(* CODESYS project HowToUse_MIC7001_baselib.2020.0527.1.project

Project tree, tasks and I/O mapping:
  Device : Changsha-Cyber-MI-linux, Changsha Cyber-MI Co., Ltd., version 3.5.10.40
    application Application
      libraries: Standard, * (System); SysFile, 3.5.15.0 (System); SysTypes2 Interfaces, * (System); SysShm, * (System); CAA Mathematics, * (CAA Technical Workgroup); SysTime, 3.5.9.0 (System); CAA Types Extern, 3.5.13.0 (CAA Technical Workgroup); CAA DTUtil Extern, 3.5.12.0 (CAA Technical Workgroup); Util, * (System); TCP, 3.5.15.0 (3S - Smart Software Solutions GmbH); CAA Net Base Services, 3.5.15.0 (CAA Technical Workgroup); MIC7001 base library, 0.93 (Cyber-MI.com); CAA SerialCom, 3.5.15.0 (CAA Technical Workgroup)
      task task_fast (cyclic, interval 20 ms, priority 10, watchdog 300 ms x 10) calls prg_data2file, prg_others
      task task_middle (cyclic, interval 100 ms, priority 20, watchdog 500 ms x 5) calls prg_mqtt
      task task_slow (cyclic, interval 500 ms, priority 30, watchdog 900 ms x 10) calls prg_retain, prg_set_inmode
      Enums/
        data type ERROR
        data type MQTT_STATE
        data type UDP_STATE_1
      data type UDP_STATE
      programs/
        program prg_set_inmode [CFC]
        program prg_data2file [ST]
        program prg_retain [ST]
        program prg_mqtt [CFC]: ACT_boot, ACT_publish, ACT_recv_proc, ACT_first_buffer, ACT_normal_buffer, ACT_running_light, proc_get_command, proc_set_command, find_key
        program prg_others [ST]
    SoftMotion General Axis Pool
    IoDrvMIC7001 : IoDrvMIC7001, Cyber-MI, version 19.1.1
        output Application.prg_others.ao_00 : DWORD  // Ao00-Ai46@C22
        output Application.prg_others.ao_01 : DWORD  // Ao01-Ai47@D14
        output Application.prg_others.led_run : BOOL  // LED_run
        output Application.prg_others.led_run : BOOL  // LED_usr
        unmapped channels: Ai00@C16, Ai01@C28, Ai02@C17, Ai03@C29, Ai04@C30, Ai05@C19, Ai06@C31, Ai07@C20, Ai08@C18, Ai09@D18, Ai10@D20, Ai11@D31, Ai12@D19, Ai13@D30, Ai14@D29, Ai15@D17, Ai16@D28, Ai17@D16, Ai18-Do00@C25, Ai19-Do01@C24, Ai20-Do02@C13, Ai21-Do03@C01, Ai22-Do04@C03, Ai23-Do05@C04, Ai24-Do06@C05, Ai25-Do07@C06, Ai26-Do08@C08, Ai27-Do09@C09, Ai28-Do10@C10, Ai29-Do11@C11, Ai30-Do12@D34, Ai31-Do13@D35, Ai32-Do14@D23, Ai33-Do15@D12, Ai34-Do16@D10, Ai35-Do17@D09, Ai36-Do18@D08, Ai37-Do19@D07, Ai38-Do20@D05, Ai39-Do21@D04,
          Ai40-Do22@D03, Ai41-Do23@D02, Ai42-Do24@C23, Ai43-Do25@C35, Ai44-Do26@D24, Ai45-Do27@D13, Ai46-Ao00@C22, Ai47-Ao01@D14, Ai48_Pi02, Ai49_Out5V, Ai50_VCC, Ai51_VCC_L, Ai52_VCC_R, Ai53_Pwm-i0, Ai54_Pwm-i1, Ai55_Pwm-i2, Ai56_Pwm-i3, Ai57_CPU-T, Ai58_G-x, Ai59_G-y, Ai60_G-z, Ai61-reserved, Ai62-IO-cntr, Ai63-CDS-cntr, Di00-Ai00@C16, Di01-Ai01@C28, Di02-Ai02@C17, Di03-Ai03@C29, Di04-Ai04@C30, Di05-Ai05@C19, Di06-Ai06@C31, Di07-Ai07@C20, Di08-Ai08@C18, Di09-Ai09@D18, Di10-Ai10@D20, Di11-Ai11@D31, Di12-Ai12@D19, Di13-Ai13@D30, Di14-Ai14@D29, Di15-Ai15@D17,
          Di16-Ai16@D28, Di17-Ai17@D16, Di18-Ai18@C25, Di19-Ai19@C24, Di20-Ai20@C13, Di21-Ai21@C01, Di22-Ai22@C03, Di23-Ai23@C04, Di24-Ai24@C05, Di25-Ai25@C06, Di26-Ai26@C08, Di27-Ai27@C09, Di28-Ai28@C10, Di29-Ai29@C11, Di30-Ai30@D34, Di31-Ai31@D35, Di32-Ai32@D23, Di33-Ai33@D12, Di34-Ai34@D10, Di35-Ai35@D09, Di36-Ai36@D08, Di37-Ai37@D07, Di38-Ai38@D05, Di39-Ai39@D04, Di40-Ai40@D03, Di41-Ai41@D02, Di42-Ai42@C23, Di43-Ai43@C35, Di44-Ai44@D24, Di45-Ai45@D13, Di46-Ai46@C22, Di47-Ai47@D14, Di48-Pi00@C15, Di49-Pi01@C14, Di50-Pi02@D22, Di51-Pi03@D21, Di52-reserved, Di53-reserved, Di54-reserved, Di55-reserved,
          Di56-reserved, Di57-reserved, Di58-reserved, Di59-reserved, Di60-reserved, Di61-reserved, Di62-reserved, Di63-reserved, Pi00-Di48@C15, Pi01-Di49@C14, Pi02-Di50@D22, Pi03-Di51@D21, Do00-Ai18@C25, Do01-Ai19@C24, Do02-Ai20@C13, Do03-Ai21@C01, Do04-Ai22@C03, Do05-Ai23@C04, Do06-Ai24@C05, Do07-Ai25@C06, Do08-Ai26@C08, Do09-Ai27@C09, Do10-Ai28@C10, Do11-Ai29@C11, Do12-Ai30@D34, Do13-Ai31@D35, Do14-Ai32@D23, Do15-Ai33@D12, Do16-Ai34@D10, Do17-Ai35@D09, Do18-Ai36@D08, Do19-Ai37@D07, Do20-Ai38@D05, Do21-Ai39@D04, Do22-Ai40@D03, Do23-Ai41@D02, Do24-Ai42@C23, Do25-Ai43@C35, Do26-Ai44@D24, Do27-Ai45@D13,
          Do28-Pwmi00@C33, Do29-Pwmi01@C34, Do30-Pwmi02@D25, Do31-Pwmi03@D26, PWM00@C25, PWM01@C24, PWM02@C13, PWM03@C01, PWM04@C03, PWM05@C04, PWM06@C05, PWM07@C06, PWM08@C08, PWM09@C09, PWM10@C10, PWM11@C11, PWM12@D34, PWM13@D35, PWM14@D23, PWM15@D12, PWM16@D10, PWM17@D09, PWM18@D08, PWM19@D07, PWM20@D05, PWM21@D04, PWM22@D03, PWM23@D02, PWM24@C23, PWM25@C35, PWM26@D24, PWM27@D13, PWM28-Pwmi00@C33, PWM29-Pwmi01@C34, PWM30-Pwmi02@D25, PWM31-Pwmi03@D26, PWM_I_0@C33, PWM_I_1@C34, PWM_I_2@D25, PWM_I_3@D26,
          LED_err, ctrl_ai_raw, ctrl_adjust, ctrl_adj0, ctrl_adj1, ctrl_adj2, ctrl_adj3, disable_5V
  libraries: VisuSymbols, 3.5.10.0 (System)
  5ce3da45-db07-42e7-a21c-a00fff4ed8f6|C:\Users\zhou\p01.bmp
  5ce3da45-db07-42e7-a21c-a00fff4ed8f6|C:\working\p01.bmp
  5ce3da45-db07-42e7-a21c-a00fff4ed8f6|C:\working\file.bmp
  text list GlobalTextList
*)

// Device/Application/UDP_STATE
TYPE UDP_STATE :
(
	INIT := 0, 	(* first State. Connections are set up *)
	SEND,		(* Send messages *)
	READ,		(* Receive messages *)
	ERROR		(* Prepare to reset connections *)
);
END_TYPE

// Device/Application/Enums/ERROR
{attribute 'qualified_only'}
//{attribute 'conditionalshow'}
//{attribute 'conditionalshow' := 'SomeText'}
//{attribute 'hide'}
TYPE ERROR : (NO_ERROR, TIME_OUT); END_TYPE

// Device/Application/Enums/MQTT_STATE
{attribute 'qualified_only'}
{attribute 'strict'}
TYPE MQTT_STATE :
(
	INIT := 0,
	CONN_SEND,
	CONN_RECV,
	READY,
	SEND,
	RECV,
	ERROR
);
END_TYPE

// Device/Application/Enums/UDP_STATE_1
TYPE UDP_STATE_1 :
(
	INIT := 0, 	(* first State. Connections are set up *)
	SEND,		(* Send messages *)
	READ,		(* Receive messages *)
	ERROR		(* Prepare to reset connections *)
);
END_TYPE

// Device/Application/programs/prg_data2file
PROGRAM prg_data2file
VAR
	data:ARRAY[0..MIC7001_base.Constants.FILE_DATA_MAX] OF REAL;
	data2file :MIC7001_base.FB_DATA2FILE;
END_VAR


data2file.xEnable := TRUE;

data[0] := 12345;  //发动机转速
data[1] := 33333;  //主泵压力
data[2] := 44444;  //液压油温
data[3] := 55555;  //油门旋钮
data[4] := 66666;  //燃油油位

data[6] := 88888;  //所有开关量

data2file(data := data, length := 70, interval := T#200MS, filedir := '/userdata/', maxsize_m := 100);

END_PROGRAM

// Device/Application/programs/prg_others
PROGRAM prg_others
VAR
	booted :BOOL := FALSE;
	mysn:STRING(32);
	
	ton_run:ton;
	led_run : BOOL := TRUE;
	
	ao_00_in:DWORD := 1234;
	ao_01_in:DWORD := 6000;
	
	ao_00:DWORD;  // 需要绑定到AO端口表中
	ao_01:DWORD;  // 需要绑定到AO端口表中
	ao_adj:mic7001_base.FB_AO_ADJ;  
	
	iccid:STRING(32);
	lac:STRING(8);
	cid:STRING(8);
	
	ton_mins:ton;
	r_mins:DINT;  //运行时间 分钟数
END_VAR


IF NOT booted THEN
	booted := TRUE;
	mic7001_base.set_piv01(6000);  //将 PI-00， PI-01的门槛电压设置为6V
	mic7001_base.set_piv23(8700);  //将 PI-02,  PI-03的门槛电压设置为8.7V
	
	mic7001_base.Disable_120ohm_can0();  //禁用CAN0口的内部终端电阻
	mic7001_base.Enable_120ohm_can1();  //启用CAN1口的内部终端电阻
	
	mic7001_base.read_sn(ADR(mysn));  //读取控制器序列号
	
	mic7001_base.set_pwm_frequency(0, 150);   //设置 C端口所有PWM频率为 150Hz  （范围： 50 ~  1000 Hz）
	mic7001_base.set_pwm_frequency(1, 300);   //设置 D端口所有PWM频率为 300Hz  （范围： 50 ~  1000 Hz）
	
	mic7001_base.read_iccid(iccid := ADR(iccid));    // 读取内部sim卡号，可作为控制器唯一标识
	mic7001_base.read_location(lac := ADR(lac), ci := ADR(cid));  //读取 GSM网络的小区号和基站号， 可通过 lbs-sir 公众号 ，输入 这两个数字查询地理位置
	r_mins := mic7001_base.read_work_mins();  // 读取控制器累计运行分钟数
END_IF

ton_mins(in := NOT ton_mins.Q, pt := T#60S);
IF ton_mins.Q THEN
	r_mins := mic7001_base.read_work_mins();  // 读取控制器累计运行分钟数
END_IF

 //运行灯 每秒闪烁一次运行灯
ton_run(in := NOT ton_run.Q, pt := T#0.5S); 
IF ton_run.Q THEN
	led_run := NOT led_run;
END_IF

// 使用 AO 端口的校准参数
ao_adj(xEnable := TRUE, in_ao_00_mv := ao_00_in, in_ao_01_mv := ao_01_in, out_ao_00 => ao_00, out_ao_01 => ao_01, xErr =>);

END_PROGRAM

// Device/Application/programs/prg_mqtt
PROGRAM prg_mqtt

VAR
	FB_MQTTClient_0: mic7001_base.FB_MQTTClient;
	
	//topic : STRING(255) := '/sys/a1SB8J9cA4L/CMI010319120011/thing/model/up_raw';
	//topic : STRING(255) := '/a1SB8J9cA4L/CMI010319120011/user/to_app';
	payload : STRING(255) := '{"RPM": 1234, "Hours": 2345}';
	
	//subscribe : STRING(255) := '/a1SB8J9cA4L/CMI010319120011/user/from_app';
	
	xPub : BOOL := FALSE;
	xSub : BOOL := FALSE;
	xBooted :BOOL := FALSE;
	
	ton_pub : ton;
	
	val_payload:ARRAY[0..32] OF mic7001_base.dut_json;
	rpm_value : DINT := 1000;
	hours_value :REAL := 680;
	time_value : STRING;
	sn_value : STRING(128);
	lac_str:STRING(128);
	cid_str:STRING(128);
	press_value :REAL := 20.1;
	
	recv_data : ARRAY[0..32] OF mic7001_base.DUT_json;
	old_recv_cntr:UDINT := 0;
	payload_len :INT;
	
	mqtt_first :BOOL := TRUE;
	ton_running:ton:=(pt := T#500MS);
	led_run:BOOL := FALSE;
	led_err:BOOL := FALSE;
	led_usr:BOOL := FALSE;
	pkg_id :DINT := 0;
	i :DINT;
	hour_today:REAL := 2.0;
	
	xLock_cmd : BOOL := FALSE;
	diLock_grade : DINT := 0;
	diLock_delay : DINT := 0;
	mqtt_interval : DINT := 5;  //mqtt package interval of publish to server	
	cntr_wait_sub : INT := 0;
END_VAR

VAR CONSTANT
	TYPE_DINT:UINT := 0;
	TYPE_REAL:UINT := 1;
	TYPE_STRING:UINT := 2;
END_VAR

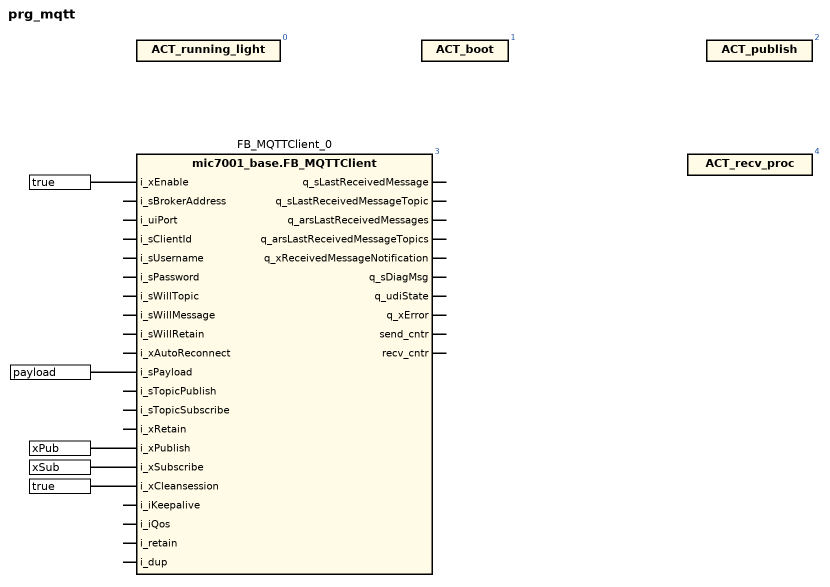
ACT_running_light();
ACT_boot();
ACT_publish();
FB_MQTTClient_0(
    i_xEnable := true,
    i_sPayload := payload,
    i_xPublish := xPub,
    i_xSubscribe := xSub,
    i_xCleansession := true); // mic7001_base.FB_MQTTClient
ACT_recv_proc();

ACTION ACT_boot:
IF NOT xbooted THEN
	IF FB_MQTTClient_0.q_udiState = 60 THEN
		xSub := TRUE;
		xBooted := TRUE;
	END_IF
END_IF
END_ACTION

ACTION ACT_publish:
IF FB_MQTTClient_0.q_udiState <> 60 THEN   //not ready, return and wait
	xPub := FALSE;
	RETURN;
END_IF

cntr_wait_sub := cntr_wait_sub + 1;
IF cntr_wait_sub < 10 THEN   // wait for subscribe succeed
	RETURN;
END_IF

IF mqtt_first THEN
	mqtt_first := FALSE;
	ACT_first_buffer();
	FB_MQTTClient_0.i_register := TRUE;
	xPub := TRUE;
	RETURN;
END_IF

ton_pub(in := NOT ton_pub.Q, pt := ANY_TO_TIME(mqtt_interval*1000));   // second to ms
IF ton_pub.Q THEN
	ACT_normal_buffer();
	FB_MQTTClient_0.i_register := FALSE;
	xPub := TRUE;
ELSE
	xPub := FALSE;
END_IF
END_ACTION

ACTION ACT_recv_proc:
(*
	cmd:  	set, get          			//命令字, set:设置参数或者执行命令，  get：点播数据或参数
	act:  	lock, unlock, reboot		//动作类型
	grade:  1, 2, 3, 4					//动作级别
	delay:  0, 60, 3600					//延迟时间,单位： 秒
*)

IF old_recv_cntr = FB_MQTTClient_0.recv_cntr THEN  //no new message
	RETURN;
END_IF
old_recv_cntr := FB_MQTTClient_0.recv_cntr;

payload_len := mic7001_base.json2arr(json := FB_MQTTClient_0.q_sLastReceivedMessage, pArr := ADR(recv_data), max_len := 32);
IF payload_len = 0 THEN
	RETURN;
END_IF

i := find_key(key := 'cmd');
IF i >= 0 AND recv_data[i].val_tp = mic7001_base.Constants.TYPE_STRING THEN 
	IF  recv_data[i].value_str = 'get' THEN
		proc_get_command();
	ELSIF recv_data[i].value_str = 'set' THEN
		proc_set_command();
	END_IF
END_IF
END_ACTION

ACTION ACT_first_buffer:

val_payload[0].key := 'sn';
val_payload[0].val_tp := TYPE_STRING;
IF MIC7001_base.read_sn(ADR(sn_value)) THEN
	val_payload[0].value_str := sn_value;
ELSE
	val_payload[0].value_str := 'SN Error';
END_IF

val_payload[1].key := 'lac';
val_payload[1].val_tp := TYPE_STRING;

val_payload[2].key := 'cid';
val_payload[2].val_tp := TYPE_STRING;

IF MIC7001_base.read_location(lac := ADR(lac_str), ci := ADR(cid_str)) THEN
	val_payload[1].value_str := lac_str; 
	val_payload[2].value_str := cid_str; 
ELSE
	val_payload[1].value_str := 'lac_error'; 
	val_payload[2].value_str := 'cid_error'; 
END_IF

val_payload[3].key := 'work_mins';
val_payload[3].val_tp := TYPE_DINT;
val_payload[3].value_dint := MIC7001_base.read_work_mins();

payload := mic7001_base.arr2json(arr := val_payload, num := 4);
END_ACTION

ACTION ACT_normal_buffer:

val_payload[0].key := 'rpm';
val_payload[0].val_tp := mic7001_base.Constants.TYPE_DINT; 
rpm_value := rpm_value + 8;
IF rpm_value > 2200 THEN
	rpm_value := 1000;
END_IF
val_payload[0].value_dint := rpm_value; 

val_payload[1].key := 'hour_all';
val_payload[1].val_tp := mic7001_base.Constants.TYPE_REAL;
hours_value := hours_value +  ANY_TO_REAL(mqtt_interval)/3600;
val_payload[1].value_real := hours_value; 

val_payload[2].key := 'power';
val_payload[2].val_tp := mic7001_base.Constants.TYPE_REAL;  
val_payload[2].value_real := ANY_TO_REAL(rpm_value)/10.0 - 39.0; 

val_payload[3].key := 'press';
val_payload[3].val_tp := mic7001_base.Constants.TYPE_REAL;  
press_value := ANY_TO_REAL(rpm_value)*1.5/100;
IF press_value > 35 THEN
	press_value := 35;
ELSIF press_value < 2 THEN
	press_value := 2;
END_IF
val_payload[3].value_real := press_value; 

val_payload[4].key := 'fuel_all';
val_payload[4].val_tp := mic7001_base.Constants.TYPE_REAL;  
val_payload[4].value_real := ANY_TO_REAL(hours_value)*13.2; 

val_payload[5].key := 'fuel_rate';
val_payload[5].val_tp := mic7001_base.Constants.TYPE_REAL; 
val_payload[5].value_real := press_value/9.1; 

val_payload[6].key := 'work_all';
val_payload[6].val_tp := mic7001_base.Constants.TYPE_REAL;
val_payload[6].value_real := hours_value*97.2; 

val_payload[7].key := 'hour_today';
val_payload[7].val_tp := mic7001_base.Constants.TYPE_REAL;
hour_today := hour_today + ANY_TO_REAL(mqtt_interval)/3600;
IF hour_today > 9 THEN
	hour_today := 2.0;
END_IF
val_payload[7].value_real := hour_today; 


val_payload[8].key := 'fuel_today';
val_payload[8].val_tp := mic7001_base.Constants.TYPE_REAL;
val_payload[8].value_real := hour_today*12.3; 

val_payload[9].key := 'work_today';
val_payload[9].val_tp := mic7001_base.Constants.TYPE_REAL;
val_payload[9].value_real := hour_today*97.2; 


payload := mic7001_base.arr2json(arr := val_payload, num := 10);
END_ACTION

ACTION ACT_running_light:
ton_running(in := NOT ton_running.Q);
IF ton_running.Q THEN
	led_run := NOT led_run;
	led_usr := FALSE;
END_IF

IF FB_MQTTClient_0.q_udiState <> 60 THEN
	led_usr := TRUE;
END_IF
END_ACTION

ACTION proc_get_command:
(*
	cmd:  	get  	//命令字, get：点播数据或参数
	rpm:  	15		//点播转速， 上传15次
	press:  0		//点播压力， 持续上传
	fuel_all: 1	  	//点播总油耗，上传一次 					
*)
END_ACTION

ACTION proc_set_command:
(*
	cmd:  	set  	          	//命令字, set:设置参数或者执行命令，  get：点播数据或参数
	interval:	15				//设置上传间隔： 15秒
	act:  	lock, unlock		//锁机动作类型
	grade:  1, 2, 3, 4			//动作级别
	delay:  0, 60, 3600			//延迟时间,单位： 秒
*)

// check lock command 
i := find_key(key := 'act');
IF i >= 0 AND recv_data[i].val_tp = mic7001_base.Constants.TYPE_STRING  THEN
	IF recv_data[i].value_str = 'lock' THEN
		xlock_cmd := TRUE;
	ELSIF recv_data[i].value_str = 'unlock' THEN
		xlock_cmd := FALSE;
	END_IF
END_IF

i := find_key(key := 'grade');
IF i >= 0 AND recv_data[i].val_tp = mic7001_base.Constants.TYPE_DINT THEN
	diLock_grade := recv_data[i].value_dint;
END_IF

i := find_key(key := 'delay');
IF i >= 0 AND recv_data[i].val_tp = mic7001_base.Constants.TYPE_DINT THEN
	diLock_delay := recv_data[i].value_dint;
END_IF

i := find_key(key := 'interval');
IF i >= 0 AND recv_data[i].val_tp = mic7001_base.Constants.TYPE_DINT THEN
	mqtt_interval := recv_data[i].value_dint;
END_IF
END_ACTION

METHOD find_key : dint
VAR_INPUT
	key :STRING(32);
END_VAR
VAR
	i :UINT;
END_VAR
find_key := -1;

FOR i := 0 TO payload_len-1 DO
	IF key = recv_data[i].key THEN
		find_key := i;
		RETURN;
	END_IF
END_FOR

RETURN; // not find,  return -1
END_METHOD

END_PROGRAM

// Device/Application/programs/prg_retain
PROGRAM prg_retain
VAR
	inited:BOOL := FALSE;
	
	// 每组retain变量可以保存100个参数，如果不够，可创建第二个
	// 下面的retain.txt.01 这个名字最好修改成其它的，避免跟其它机型重复，造成售后万一调换控制器后参数混淆
	myRetain01:mic7001_base.FB_RETAIN := (filename := '/userdata/retain.txt.01', use_bak := TRUE);  
	//retain 变量, 建议放在全局变量列表 gvl中
	g_retain01:ARRAY[0..mic7001_base.Constants.RETAIN_NUM_MAX] OF DINT;
	
	// 如果上面的100个参数不够用，可以打开下面这两行的注释 ，增加另外100个
(*	myRetain02:mic7001_base.FB_RETAIN := (filename := '/userdata/retain.txt.02', use_bak := TRUE);
	g_retain02:ARRAY[0..mic7001_base.Constants.RETAIN_NUM_MAX] OF DINT;	
*)	
	



END_VAR

//步骤一：初始化默认值,如果读取文件失败，则使用默认值作为当前参数
IF NOT inited THEN  //上电执行一次，设置retain变量的缺省值
	//第一组retain变量初始值，新控制器第一次上电有效。
	myRetain01.default_val[0] := 123;
	myRetain01.default_val[1] := 456;
	myRetain01.default_val[2] := 789;
	// .....
	myRetain01.default_val[87] := 321;
	myRetain01.default_val[99] := 1234;  //最后一个

	//第二组retain变量初始值，新控制器第一次上电有效。
(*	myRetain02.default_val[0] := 999;
	myRetain02.default_val[1] := 888;
	myRetain02.default_val[2] := 777;
	// .....
	myRetain02.default_val[98] := 333;
	myRetain02.default_val[99] := 222;  //最后一个
*)	
	inited := TRUE;
END_IF

//步骤二：执行功能块，处理参数的保存和读取
myRetain01(value := g_retain01);
(*
myRetain02(value := g_retain02);
*)

//步骤三：在其它任务中直接使用 g_retain01[]   和 g_retain02[] 作为retain变量

END_PROGRAM

// Device/Application/programs/prg_set_inmode
PROGRAM prg_set_inmode
VAR
	FB_SET_INMODE_0: MIC7001_BASE.FB_SET_INMODE;
END_VAR

VAR CONSTANT
	MODE_5V: 	UINT := 0;
	MODE_36V:	UINT := 1;
	MODE_20mA:	UINT := 2;
	MODE_30K : 	UINT := 3;
	MODE_DI_H: 	UINT := 4;
	MODE_DI_L: 	UINT := 5;
END_VAR

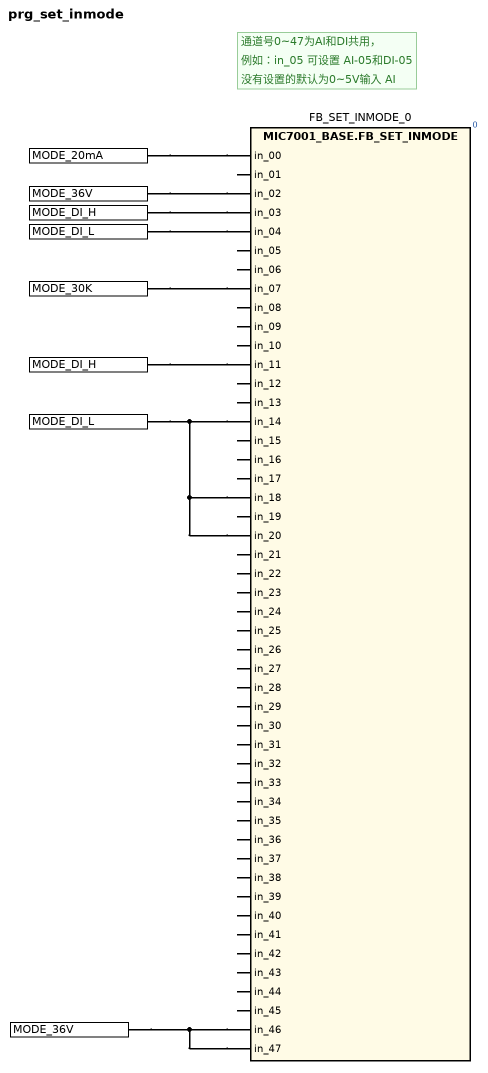
// 通道号0~47为AI和DI共用，
// 例如：in_05 可设置 AI-05和DI-05
// 没有设置的默认为0~5V输入 AI
FB_SET_INMODE_0(
    in_00 := MODE_20mA,
    in_02 := MODE_36V,
    in_03 := MODE_DI_H,
    in_04 := MODE_DI_L,
    in_07 := MODE_30K,
    in_11 := MODE_DI_H,
    in_14 := MODE_DI_L,
    in_18 := MODE_DI_L,
    in_20 := MODE_DI_L,
    in_46 := MODE_36V,
    in_47 := MODE_36V); // MIC7001_BASE.FB_SET_INMODE

END_PROGRAM
